// Device/Application/MANUAL_FRAME_1
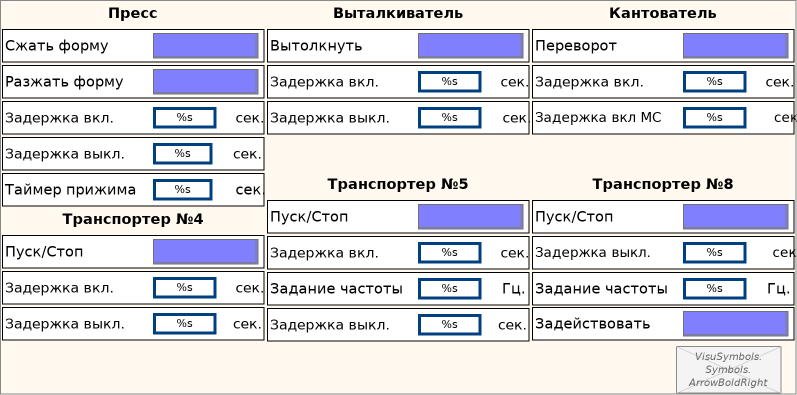
VISUALIZATION MANUAL_FRAME_1  // 797x395
    Rectangle (2,29 262x33), "Сжать форму"
    Rectangle (2,65 262x33), "Разжать форму"
    Rectangle (2,2 262x22), "Пресс"
    Button (153,33 105x25), colour toggle: GVL.XV01KV207_MANOI
        OnMouseClick:  ToggleVariable=GVL.XV01KV207_MANOI
    Button (153,69 105x25), colour toggle: GVL.XV02KV208_MANOI
        OnMouseClick:  ToggleVariable=GVL.XV02KV208_MANOI
    Rectangle (267,29 262x33), "Вытолкнуть"
    Rectangle (267,2 262x22), "Выталкиватель"
    Button (418,33 105x25), colour toggle: GVL.XV03KV209_MANOI
        OnMouseClick:  ToggleVariable=GVL.XV03KV209_MANOI
    Rectangle (532,29 262x33), "Переворот"
    Rectangle (532,65 262x33), "Задержка вкл. сек."
    Rectangle (532,2 262x22), "Кантователь"
    Button (683,33 105x25), colour toggle: GVL.M07KM07_MANOI
        OnMouseClick:  ToggleVariable=GVL.M07KM07_MANOI
    Rectangle (683,71 63x21), "%s", text variable: GVLR.TIME_M07KM07_DELAY
        OnMouseClick: write the text variable via VisuDialogs.Numpad
    Rectangle (2,101 262x33), "Задержка вкл. сек."
    Rectangle (153,107 63x21), "%s", text variable: GVLR.TIME_XV01KV207_DELAY
        OnMouseClick: write the text variable via VisuDialogs.Numpad
    Rectangle (2,137 262x33), "Задержка выкл. сек."
    Rectangle (153,143 59x21), "%s", text variable: GVLR.TIME_XV02KV208_DELAY
        OnMouseClick: write the text variable via VisuDialogs.Numpad, min 0, max 5
    Rectangle (267,65 262x33), "Задержка вкл. сек."
    Rectangle (418,71 63x21), "%s", text variable: GVLR.TIME_XV03KV209_DELAY
        OnMouseClick: write the text variable via VisuDialogs.Numpad
    Rectangle (267,101 262x33), "Задержка выкл. сек."
    Rectangle (418,107 63x21), "%s", text variable: GVLR.TIME_XV03KV209_UP
        OnMouseClick: write the text variable via VisuDialogs.Numpad, min 1
    Rectangle (2,235 262x33), "Пуск/Стоп"
    Rectangle (2,271 262x33), "Задержка вкл. сек."
    Rectangle (2,208 262x22), "Транспортер №4"
    Button (153,239 105x25), colour toggle: GVL.M08KM08_MANOI
        OnMouseClick:  ToggleVariable=GVL.M08KM08_MANOI
    Rectangle (153,277 63x21), "%s", text variable: GVLR.TIME_M08KM08_DELAY
        OnMouseClick: write the text variable via VisuDialogs.Numpad
    Rectangle (267,200 262x33), "Пуск/Стоп"
    Rectangle (267,236 262x33), "Задержка вкл. сек."
    Rectangle (267,173 262x22), "Транспортер №5"
    Button (418,204 105x25), colour toggle: GVL.M09UZ09_MANOI
        OnMouseClick:  ToggleVariable=GVL.M09UZ09_MANOI
    Rectangle (267,272 262x33), "Задание частоты Гц."
    Rectangle (418,278 63x21), "%s", text variable: GVLR.M09UZ09_SP
        OnMouseClick: write the text variable via VisuDialogs.Numpad
    Rectangle (418,242 63x21), "%s", text variable: GVLR.TIME_M09UZ09_DELAY
        OnMouseClick: write the text variable via VisuDialogs.Numpad
    Rectangle (532,200 262x33), "Пуск/Стоп"
    Rectangle (532,236 262x33), "Задержка выкл. сек."
    Rectangle (532,173 262x22), "Транспортер №8"
    Button (683,204 105x25), colour toggle: GVL.M14UZ14_MANOI
        OnMouseClick:  ToggleVariable=GVL.M14UZ14_MANOI
    Rectangle (532,272 262x33), "Задание частоты Гц."
    Rectangle (683,278 63x21), "%s", text variable: GVLR.M14UZ14_SP
        OnMouseClick: write the text variable via VisuDialogs.Numpad
    Rectangle (683,242 63x21), "%s", text variable: GVLR.TIME_M14UZ14_OFF
        OnMouseClick: write the text variable via VisuDialogs.Numpad
    Image (676,346 105x47), image: VisuSymbols.Symbols.ArrowBoldRight
        OnMouseClick: FrameSelectionChange Selection=Selection=-1, GlobSel=IndExpr=7, AssignDir=Main.GenElemInst_39, AssignType=Directly, SelType=Globally
    Rectangle (267,308 262x33), "Задержка выкл. сек."
    Rectangle (418,314 63x21), "%s", text variable: GVLR.TIME_M09UZ09_OFF
        OnMouseClick: write the text variable via VisuDialogs.Numpad
    Rectangle (532,307 262x33), "Задействовать"
    Button (683,311 105x25), colour toggle: GVL.M14UZ14_CFGOI
        OnMouseClick:  ToggleVariable=GVL.M14UZ14_CFGOI
    Rectangle (2,307 262x33), "Задержка выкл. сек."
    Rectangle (153,313 63x21), "%s", text variable: GVLR.TIME_M08KM08_OFF
        OnMouseClick: write the text variable via VisuDialogs.Numpad
    Rectangle (532,101 262x33), "Задержка вкл МС сек."
    Rectangle (683,107 63x21), "%s", text variable: GVLR.TIME_SPEED2_DELAY
        OnMouseClick: write the text variable via VisuDialogs.Numpad, min 0, max 3
    Rectangle (2,173 262x33), "Таймер прижима сек."
    Rectangle (153,179 59x21), "%s", text variable: GVLR.TIMER_SQ5_DELAY
        OnMouseClick: write the text variable via VisuDialogs.Numpad, min 0.1, max 5
END_VISUALIZATION

// Device/Application/MANUAL_FRAME_2
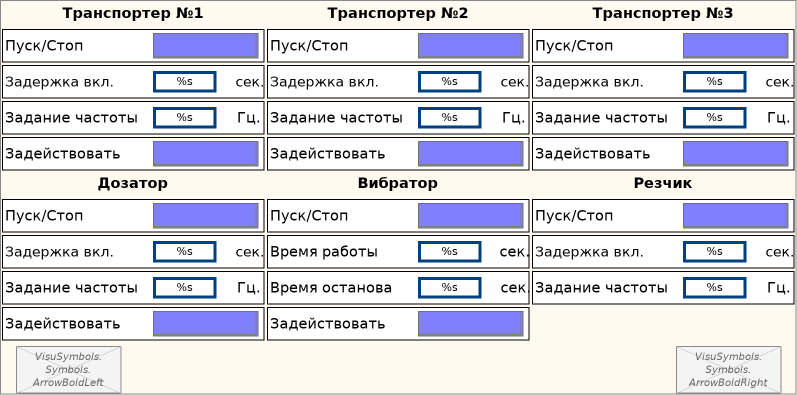
VISUALIZATION MANUAL_FRAME_2  // 797x395
    Rectangle (2,29 262x33), "Пуск/Стоп"
    Rectangle (2,2 262x22), "Транспортер №1"
    Button (153,33 105x25), colour toggle: GVL.M03UZ03_MANOI
        OnMouseClick:  ToggleVariable=GVL.M03UZ03_MANOI
    Rectangle (2,65 262x33), "Задержка вкл. сек."
    Rectangle (153,71 63x21), "%s", text variable: GVLR.TIME_M03UZ03_DELAY
        OnMouseClick: write the text variable via VisuDialogs.Numpad
    Rectangle (2,101 262x33), "Задание частоты Гц."
    Rectangle (153,107 63x21), "%s", text variable: GVLR.M03UZ03_SP
        OnMouseClick: write the text variable via VisuDialogs.Numpad
    Rectangle (267,29 262x33), "Пуск/Стоп"
    Rectangle (267,2 262x22), "Транспортер №2"
    Button (418,33 105x25), colour toggle: GVL.M05UZ05_MANOI
        OnMouseClick:  ToggleVariable=GVL.M05UZ05_MANOI
    Rectangle (267,65 262x33), "Задержка вкл. сек."
    Rectangle (418,71 63x21), "%s", text variable: GVLR.TIME_M05UZ05_DELAY
        OnMouseClick: write the text variable via VisuDialogs.Numpad
    Rectangle (267,101 262x33), "Задание частоты Гц."
    Rectangle (418,107 63x21), "%s", text variable: GVLR.M05UZ05_SP
        OnMouseClick: write the text variable via VisuDialogs.Numpad
    Rectangle (532,29 262x33), "Пуск/Стоп"
    Rectangle (532,2 262x22), "Транспортер №3"
    Button (683,33 105x25), colour toggle: GVL.M06UZ06_MANOI
        OnMouseClick:  ToggleVariable=GVL.M06UZ06_MANOI
    Rectangle (532,65 262x33), "Задержка вкл. сек."
    Rectangle (683,71 63x21), "%s", text variable: GVLR.TIME_M06UZ06_DELAY
        OnMouseClick: write the text variable via VisuDialogs.Numpad
    Rectangle (532,101 262x33), "Задание частоты Гц."
    Rectangle (683,107 63x21), "%s", text variable: GVLR.M06UZ06_SP
        OnMouseClick: write the text variable via VisuDialogs.Numpad
    Rectangle (2,199 262x33), "Пуск/Стоп"
    Rectangle (2,172 262x22), "Дозатор"
    Button (153,203 105x25), colour toggle: GVL.M01UZ01_MANOI
        OnMouseClick:  ToggleVariable=GVL.M01UZ01_MANOI
    Rectangle (2,235 262x33), "Задержка вкл. сек."
    Rectangle (153,241 63x21), "%s", text variable: GVLR.TIME_M01UZ01_DELAY
        OnMouseClick: write the text variable via VisuDialogs.Numpad
    Rectangle (2,271 262x33), "Задание частоты Гц."
    Rectangle (153,277 63x21), "%s", text variable: GVLR.M01UZ01_SP
        OnMouseClick: write the text variable via VisuDialogs.Numpad
    Rectangle (2,307 262x33), "Задействовать"
    Rectangle (267,199 262x33), "Пуск/Стоп"
    Rectangle (267,172 262x22), "Вибратор"
    Button (418,203 105x25), colour toggle: GVL.MV01KM00_MANOI
        OnMouseClick:  ToggleVariable=GVL.MV01KM00_MANOI
    Rectangle (267,235 262x33), "Время работы сек."
    Rectangle (418,241 63x21), "%s", text variable: GVLR.TIME_MV01KM00_ON
        OnMouseClick: write the text variable via VisuDialogs.Numpad
    Rectangle (532,172 262x22), "Резчик"
    Image (16,346 105x47), image: VisuSymbols.Symbols.ArrowBoldLeft
        OnMouseClick: FrameSelectionChange Selection=Selection=-1, GlobSel=IndExpr=6, AssignDir=Main.GenElemInst_39, AssignType=Directly, SelType=Globally
    Rectangle (532,199 262x33), "Пуск/Стоп"
    Button (683,203 105x25), colour toggle: GVL.M02UZ02_MANOI
        OnMouseClick:  ToggleVariable=GVL.M02UZ02_MANOI
    Rectangle (532,235 262x33), "Задержка вкл. сек."
    Rectangle (683,241 63x21), "%s", text variable: GVLR.TIME_M02UZ02_DELAY
        OnMouseClick: write the text variable via VisuDialogs.Numpad
    Rectangle (532,271 262x33), "Задание частоты Гц."
    Rectangle (683,277 63x21), "%s", text variable: GVLR.M02UZ02_SP
        OnMouseClick: write the text variable via VisuDialogs.Numpad
    Button (153,311 105x25), colour toggle: GVL.M01UZ01_CFGOI
        OnMouseClick:  ToggleVariable=GVL.M01UZ01_CFGOI
    Rectangle (267,271 262x33), "Время останова сек."
    Rectangle (418,277 63x21), "%s", text variable: GVLR.TIME_MV01KM00_OFF
        OnMouseClick: write the text variable via VisuDialogs.Numpad
    Image (676,346 105x47), image: VisuSymbols.Symbols.ArrowBoldRight
        OnMouseClick: FrameSelectionChange Selection=Selection=-1, GlobSel=IndExpr=8, AssignDir=Main.GenElemInst_39, AssignType=Directly, SelType=Globally
    Rectangle (267,307 262x33), "Задействовать"
    Button (418,311 105x25), colour toggle: GVL.MV01KM00_CFGOI
        OnMouseClick:  ToggleVariable=GVL.MV01KM00_CFGOI
    Rectangle (532,137 262x33), "Задействовать"
    Button (683,141 105x25), colour toggle: GVL.M06UZ06_CFGOI
        OnMouseClick:  ToggleVariable=GVL.M06UZ06_CFGOI
    Rectangle (267,137 262x33), "Задействовать"
    Button (418,141 105x25), colour toggle: GVL.M05UZ05_CFGOI
        OnMouseClick:  ToggleVariable=GVL.M05UZ05_CFGOI
    Rectangle (2,137 262x33), "Задействовать"
    Button (153,141 105x25), colour toggle: GVL.M03UZ03_CFGOI
        OnMouseClick:  ToggleVariable=GVL.M03UZ03_CFGOI
END_VISUALIZATION

// Device/Application/MANUAL_FRAME_3
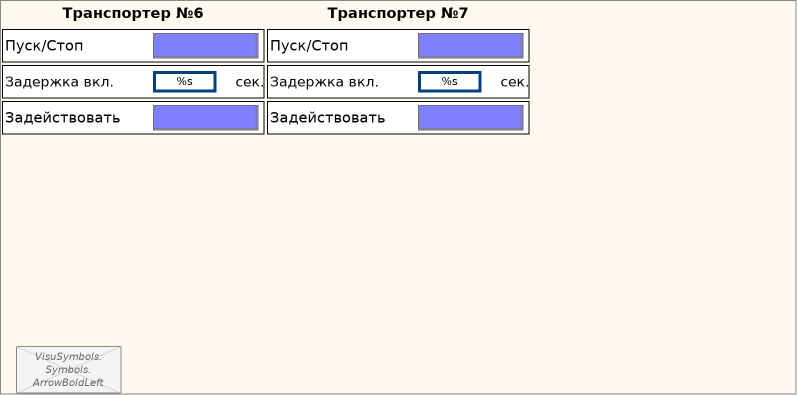
VISUALIZATION MANUAL_FRAME_3  // 797x395
    Rectangle (2,29 262x33), "Пуск/Стоп"
    Rectangle (2,2 262x22), "Транспортер №6"
    Button (153,33 105x25), colour toggle: GVL.M11KM11_MANOI
        OnMouseClick:  ToggleVariable=GVL.M11KM11_MANOI
    Rectangle (2,65 262x33), "Задержка вкл. сек."
    Rectangle (153,71 63x21), "%s", text variable: GVLR.TIME_M11KM11_DELAY
        OnMouseClick: write the text variable via VisuDialogs.Numpad
    Rectangle (267,29 262x33), "Пуск/Стоп"
    Rectangle (267,2 262x22), "Транспортер №7"
    Button (418,33 105x25), colour toggle: GVL.M12KM12_MANOI
        OnMouseClick:  ToggleVariable=GVL.M12KM12_MANOI
    Rectangle (267,65 262x33), "Задержка вкл. сек."
    Rectangle (418,71 63x21), "%s", text variable: GVLR.TIME_M12KM12_DELAY
        OnMouseClick: write the text variable via VisuDialogs.Numpad
    Image (16,346 105x47), image: VisuSymbols.Symbols.ArrowBoldLeft
        OnMouseClick: FrameSelectionChange Selection=Selection=-1, GlobSel=IndExpr=7, AssignDir=Main.GenElemInst_39, AssignType=Directly, SelType=Globally
    Rectangle (2,101 262x33), "Задействовать"
    Button (153,105 105x25), colour toggle: GVL.M11KM11_CFGOI
        OnMouseClick:  ToggleVariable=GVL.M11KM11_CFGOI
    Rectangle (267,101 262x33), "Задействовать"
    Button (418,105 105x25), colour toggle: GVL.M12KM12_CFGOI
        OnMouseClick:  ToggleVariable=GVL.M12KM12_CFGOI
END_VISUALIZATION

(* text list AlarmGroup (id | default)
  25 | Авария датчика верхнего положения выталкивателя SQ06 (геркон).
  24 | Авария транспортера №8 M14UZ14
  23 | Авария транспортера возврата обрези №7 M12KM12
  22 | Авария транспортера возврата песка №6 M11KM11
  21 | Авария транспортера №5 M09UZ09
  20 | Авария транспортера подачи рамок №4 M08KM08
  19 | Авария транспортера №3 M06UZ06
  18 | Авария транспортера №2 M05UZ05
  17 | Авария электромагнитного тормаза резчика M04KM04
  16 | Авария транспортера №1 M03UZ03
  15 | Авария резчика M02UZ02
  14 | Авария дозатора обсыпного бункера M01UZ01
  13 | Авария вибратора обсыпного бункера MV01KM00
  12 | Включен тестовый режим пресса "СЖАТЬ" XV01KV207
  11 | Превышено время ожидания на переворот кантователя SQ08
  10 | Авария маслостанции
  9 | Низкое давление масла PI01
  8 | Авария кантователя M07KM07
  7 | Превышено время ожидания на возврат выталкивателя SQ06
  6 | Превышено время ожидания на выталкивание
  5 | Превышено время ожидания на разжатие пресса SQ04
  4 | Превышено время ожидания на сжатие пресса SQ05
  3 | Отсутствует напряжение 380V QF1..QF16
  2 | Отсутствует напряжение +24V QF26
  1 | Отсутствует напряжение +24V QF25
  0 | Нажата аварийная кнопка
   |  *)

(* text list Mode (id | default)
  1 | Авто
  2 | Тест
  3 | Ручной
   |  *)

(* text list IM_TAGS (id | default)
  1 | XV01/XV02
  2 | XV03/XV04
  3 | MV01KM00
  4 | M01UZ01
  5 | M03UZ03
  6 | M04KM04
  7 | M05UZ05
  8 | M06UZ06
  9 | M07KM07
  10 | M08KM08
  11 | M09UZ09
  12 | M10KM10
  13 | M11KM11
  14 | M12KM12
  15 | M14UZ14
   |  *)

(* text list IM (id | default)
  1 | ПРФ - сжать/расжать форму
  2 | ПРФ - сжать/расжать форму
  3 | ПРФ - выталкиватель
  4 | ПРФ - выталкиватель
  5 | Вибратор обсыпн. бункера
  6 | Дозатор обсыпн. Бункера
  7 | Транспортер №1
  8 | Резчик
  9 | Транспортер №2
  10 | Транспортер №3
  11 | ПРФ - кантователь
  12 | Транспортер №4
  13 | Транспортер №5
  14 | Маслостанция
  15 | Транспортер №6
  16 | Транспортер №7
  17 | Транспортер №8
  0 | ЛИНИЯ РУЧНОЙ ФОРМОВКИ
  18 | Датчик давления масла PI01
  19 | Датчик поз. кантователя SQ08
  20 | Датчик верхнего пол. выталкивателя SQ06 (геркон)
  21 | Задержка включения малой скорости
   |  *)
